(*********************************** G.D S.p.A. - Technical Department ***********************************
============= PROGRAM INFO ============
FOLDER:             TBD
MACHINES INVOLVED:  TBD 

============= DESCRIPTION =============
csp machine declaration

============= REVISIONS ===============
Date		Version	 	Author      	Description             
----------	-------		------------  	--------------------------------------------
2019/04/05 	0000.00	 	M.Grasso		Creation of the PRG

**********************************************************************************************************)
(*$R process_ref := prc; $*)
PROGRAM csp_case_feed_arm
VAR
		
	prc:											process;
	prc_path:										STRING;
END_VAR

_read_var_input();

_object_manager();

IF NOT objects_running()
THEN
	RETURN;	
END_IF

_read_process_image();

_mode_manager();

_set_runtime_properties();

(********************************* BODY *********************************)
(************************************************************************)

_handle_messages();

_write_output();

ACTION _handle_messages:
;
END_ACTION

ACTION _handle_process_test:
;
END_ACTION

ACTION _mode_manager:
IF process_mode_req_is_pending(prc)
THEN
    process_apply_mode_req_first_step(prc);
    CASE process_get_mode(prc) OF
        MODE_TO_ABSENT:
			;
        MODE_TO_INACTIVE:
			;
        MODE_TO_TEST:
			;
        MODE_TO_OPERATIONAL:
			;
    END_CASE
    process_apply_mode_req_second_step(prc);
END_IF
END_ACTION

ACTION _object_manager:
IF objects_initialization()
THEN
	sub_process_init(
		object_name					:= 'csp_case_feed_arm.prc', 
		process						:= csp_case_feed.prc, 
		CONVERSION_this				:= prc);
		
	prc_path 						:= process_get_path(prc);
END_IF

IF objects_running()
THEN
	process_cycle(prc);
END_IF
END_ACTION

ACTION _read_process_image:
;
END_ACTION

ACTION _read_var_input:
;
END_ACTION

ACTION _set_runtime_properties:
;
END_ACTION

ACTION _write_output:
;
END_ACTION

END_PROGRAM

(* stored: Version 1.1.0.1, ProductVersion 3.1.4022.12
   POU csp_case_feed_arm: Id {a5aa59bc-22cb-47d5-9233-1014de2d77e3}, SpecialFunc None
   Action _handle_messages: Id {a93c07e7-661b-40f2-929e-fb8babe8788e}
   Action _handle_process_test: Id {d7875e82-259c-4ff1-9844-f5d378676329}
   Action _mode_manager: Id {e1ec7f07-f815-4775-8781-a309e2be1106}
   Action _object_manager: Id {8f6da173-1122-493e-8df8-ef467c219a6b}
   Action _read_process_image: Id {a493318a-a189-4da7-8830-4c383a78bddf}
   Action _read_var_input: Id {f77cf2d8-1731-47d5-acb4-b508d2bc3603}
   Action _set_runtime_properties: Id {070a85ad-8918-4546-ae4e-92df25d023e8}
   Action _write_output: Id {d4f77273-e14c-4523-ac08-c5acd7aeda86} *)
